FUNCTION_BLOCK XyTableActuatorPen EXTENDS ZEquipment.ActuatorDigitalBiLsPlusMinus

METHOD PUBLIC DownAsync
VAR_INPUT
  startToken : ZCore.IStartToken;
END_VAR
MoveMinusAsync(startToken:=startToken);
END_METHOD

METHOD PUBLIC IsDown : BOOL
VAR_INPUT
END_VAR
IsDown := IsAtMinus();
END_METHOD

METHOD PUBLIC IsUp : BOOL
VAR_INPUT
END_VAR
IsUp := IsAtPlus();
END_METHOD

METHOD PUBLIC UpAsync
VAR_INPUT
  startToken : ZCore.IStartToken;
END_VAR
MovePlusAsync(startToken:=startToken);
END_METHOD

END_FUNCTION_BLOCK

(* stored: Version 1.1.0.1
   POU XyTableActuatorPen: Id {81a3e87e-8644-49b3-b809-986ff960638c}, SpecialFunc None
   Method DownAsync: Id {2380fe05-462e-4507-8be1-c99ee40b0ee1}
   Method IsDown: Id {bc52c344-06af-4872-8b09-d92d912e03ae}
   Method IsUp: Id {37129c7a-556e-4e6b-8fbd-543b6ab9c5b3}
   Method UpAsync: Id {3c334fc2-0157-45ef-8c81-153bc3ec3ad2} *)
